// TIA Portal V20 export
TYPE "LDrive_typeKistlerPressDataSend"
// stored: IsFailsafeCompliant false
   STRUCT
      systemFixed : Struct
         Start : Bool;   // Mirrored Start Measuring
         TareY : Bool;   // Mirrored Channel Y Tare or Reset Piezo
         ZeroX : Bool;   // Mirrored Channel X zeros
         STestX : Bool;   // Mirrored Trigger sensor test for sensor X
         STestY : Bool;   // Mirrored Trigger sensor test for sensor Y
         ZeroExtendedX : Bool;
         MasterMeas : Bool;   // Mirrored Master measurement
         IncZero : Bool;   // Mirrored Zeros incremental sensor
         AckAdminGlobal : Bool;
         AckAdmin : Bool;   // Mirrored Acknowledgment with Admin rights (e.g., corresponding
         reserved1 : Bool;
         Access : Bool;   // Mirrored Allows the PLC to give the operator access rights
         Auto : Bool;   // Mirrored Auto, no editing of setup is possible
         StatReset : Bool;   // Mirrored statistics reset
         StatDisable : Bool;   // Deactivate mirrored statistics
         TaraExtendedY : Bool;
         MP : Byte;   // Mirrored measurement program choice
         reserved2 : Bool;
         reserved3 : Bool;
         resetSnGenerator : Bool;
         reserved4 : Bool;
         reserved5 : Bool;
         reserved6 : Bool;
         ExportPVTStart : Bool;
         reserved7 : Bool;
         UNI0 : Bool;   // Mirrored input signal UNI
         UNI1 : Bool;   // Mirrored input signal UNI
         UNI2 : Bool;   // Mirrored input signal UNI
         UNI3 : Bool;   // Mirrored input signal UNI
         UNI4 : Bool;   // Mirrored input signal UNI
         UNI5 : Bool;   // Mirrored input signal UNI
         UNI6 : Bool;   // Mirrored input signal UNI
         UNI7 : Bool;   // Mirrored input signal UNI
         ReservedByte1 : Byte;
         ReservedByte2 : Byte;
         ReservedByte3 : Byte;
         ReservedByte4 : Byte;
         DriveEnable : Bool;   // Mirrored enable drive
         RunSequence : Bool;   // Mirrored command process of the sequence
         DriveToHomePos : Bool;   // Mirrored command movement on base setting (MP-specific)
         DriveToRefPos : Bool;   // Mirrored command movement to reference position
         JogFW : Bool;   // Mirrored command jogging forwards
         JogBW : Bool;   // Mirrored command jogging backwards
         ContinueFromWait : Bool;   // Already
         manualBrakeTest : Bool;
         ExternalSequenceStopReq : Byte;
         ReservedByte5 : Byte;
         SelectSequence : Byte;
         ReservedByte6 : Byte;
         Cfg_MP : Byte;   // Mirrored measurement program choice of the input telegram
         jogToPosition : Bool;
         Reserved15 : Bool;
         Reserved16 : Bool;
         Reserved17 : Bool;
         Reserved18 : Bool;
         Reserved19 : Bool;   // Mirrored bit of the input telegram
         Reserved20 : Bool;   // Mirrored bit of the input telegram
         Reserved21 : Bool;   // Mirrored bit of the input telegram
         CFG_ADR : Byte;   // Mirror CFG-ADR (up V 1.2.x.)
         CFG_Length : Byte;   // Mirror CFG-LENGTH (up V 1.2.x.)
         SelectedPage : Byte;   // Mirrored page select of the input telegram
         SaveToMP : Bool;
         strobe : Bool;
         Reserved22 : Bool;   // Mirrored bit of the input telegram
         Reserved23 : Bool;   // Mirrored bit of the input telegram
         resetChangeSelectedMP : Bool;
         Reserved24 : Bool;   // Mirrored bit of the input telegram
         resetChangedGlobal : Bool;
         backupRequest : Bool;
      END_STRUCT;
      userDefinedOutData : Array[20..219] of Byte;
   END_STRUCT;
END_TYPE
